{attribute addProperty BoxType "EL5152-0000-0018"}
{attribute addProperty Id "ControlAT %Q*Control_879818281620Set_counter_valueAT %Q*UINT16217"}
{attribute addProperty CRC "2987265969"}
{attribute addProperty SizeInBites "32"}
{attribute addProperty SizeInBytes "4"}
TYPE ENC_Control_compact_Channel_B20E0FB1 :
STRUCT
	{attribute addProperty Name "Control"}
	Control AT %Q* : Control_87981828;
	{attribute addProperty Name "Set_counter_value"}
	Set_counter_value AT %Q* : UINT;
END_STRUCT
END_TYPE

(* stored: Version 1.2.0.0, ProductVersion 3.1.4024.9
   DUT ENC_Control_compact_Channel_B20E0FB1: Id {7329a1ce-a8a7-4dca-a641-848b65c91bcf} *)
